INTERFACE I_MachiningOperation

METHOD Execute : BOOL
VAR_INPUT
END_VAR
END_METHOD

END_INTERFACE

(* stored: Version 1.1.0.1, ProductVersion 3.1.4024.15
   Itf I_MachiningOperation: Id {2dfc726d-310d-4ee1-8c82-278f7369c5a0}
   Method Execute: Id {a98811e5-8c7a-4cba-a643-e6cf52a96585} *)
